Fanuc KAREL source: kt00994.KL

-- PROVISIONAL review KL for V940-1; original PC SHA256 df4df306dd207cd66c060888bee8be3d0bac2168e45f3499a533bbe5e307508b
-- Incomplete behavior may be omitted. Consult companion uncertainty JSON. Do not deploy.
PROGRAM KT00994
%NOLOCKGROUP
VAR
  X : REAL
  Y : REAL
  Z : REAL
  W : REAL
  P : REAL
  R : REAL
-- UNRESOLVED_DECL P1 type=000199
-- UNRESOLVED_DECL P2 type=000199
-- UNRESOLVED_DECL CFG type=00001c
BEGIN
  -- V9_ZERO_TABLE_METADATA_HINT layout=0001; no indexed target words; source/name/runtime held
  -- UNRESOLVED_PC offsets 5-65; opcodes 27,27,49,7E,AD,22,22,22,22,22,22,22,76
  -- UNRESOLVED_PC offsets 70-74; opcodes 7F
END KT00994
